			(* Постоянная часть передачи *)
			t_Msg.t_Id.u32_Id := 16#101;		(* Адрес пакета *)
			t_Msg.t_Id.u8_Xtd := 0;
			t_Msg.u8_Dlc      := 8;				(* Количество передаваемых байт *)
			t_Msg.au8_Data[0] := Can_buffer[CAN_TX_count+1];
			t_Msg.au8_Data[1] := Can_buffer[CAN_TX_count+2];
			t_Msg.au8_Data[2] := Can_buffer[CAN_TX_count+3];
			t_Msg.au8_Data[3] := Can_buffer[CAN_TX_count+4];
			t_Msg.au8_Data[4] := Can_buffer[CAN_TX_count+5];
			t_Msg.au8_Data[5] := Can_buffer[CAN_TX_count+6];
			t_Msg.au8_Data[6] := Can_buffer[CAN_TX_count+7];
			t_Msg.au8_Data[7] := Can_buffer[CAN_TX_count+8];
			fb_CanObjSendMsg(ou32_Handle:=TX, ot_Msg:=t_Msg, os16_Status=>s16_Return);
			CAN_TX_count:=CAN_TX_count+8;
		END_IF

END_IF
END_PROGRAM

(* POU CAN/Recieve, ST *)
PROGRAM Recieve
VAR
	s16_Return        	: INT;
	r_Msg			         : T_x_can_msg;
	fb_CanObjGetMsg   	: FB_x_can_obj_get_msg;
	fb_EepWrite  			: FB_x_eep_write;

	u16_Crc           	: UINT;
	fb_UtiCalcCrc16   	: FB_x_uti_calc_crc_16;
	i: WORD; (* Счетчик принятых по CAN пакетов в калибровке *)

	crc_given: UINT;
END_VAR
IF Flag_CAN THEN
			(* Что бы при ошибке чтения с CANa , при не изменении значений не произошо ложного срабатывания *)
			r_Msg.au8_Data[0]:=0;r_Msg.au8_Data[1]:=0;r_Msg.au8_Data[2]:=0;r_Msg.au8_Data[3]:=0;r_Msg.au8_Data[4]:=0;
			r_Msg.au8_Data[5]:=0;r_Msg.au8_Data[6]:=0;r_Msg.au8_Data[7]:=0;
			fb_CanObjGetMsg(ou32_Handle:=RX, ot_Msg=>r_Msg, os16_Status=>s16_Return);
			IF s16_Return = C_NO_ERR THEN

					(* Поступил запрос на передачу? *)
					IF	Flag_CAN_recieve=FALSE AND r_Msg.au8_Data[0] = 8 AND r_Msg.au8_Data[1] = 7 AND r_Msg.au8_Data[2] = 6 AND r_Msg.au8_Data[3] = 5 AND
						r_Msg.au8_Data[4] = 4 AND r_Msg.au8_Data[5] = 3 AND r_Msg.au8_Data[6] = 2 AND	r_Msg.au8_Data[7] = 1 THEN
						Flag_CAN_send:=TRUE;
					END_IF

					(* Поступил запрос на прием ? *)
					IF Flag_CAN_recieve = FALSE AND r_Msg.au8_Data[0] = 1 AND r_Msg.au8_Data[1] = 2 AND r_Msg.au8_Data[2] = 3 AND r_Msg.au8_Data[3] = 4 AND
						r_Msg.au8_Data[4] = 5 AND r_Msg.au8_Data[5] = 6 AND r_Msg.au8_Data[6] = 7 AND r_Msg.au8_Data[7] = 8 THEN

									Flag_CAN_recieve:=TRUE;
									i:=1;
					ELSIF i <= SIZEOF(Can_buffer)-7 THEN
											Can_buffer[i]:=r_Msg.au8_Data[0]; Can_buffer[i+1]:=r_Msg.au8_Data[1]; Can_buffer[i+2]:=r_Msg.au8_Data[2]; Can_buffer[i+3]:=r_Msg.au8_Data[3];
											Can_buffer[i+4]:=r_Msg.au8_Data[4]; Can_buffer[i+5]:=r_Msg.au8_Data[5]; Can_buffer[i+6]:=r_Msg.au8_Data[6]; Can_buffer[i+7]:=r_Msg.au8_Data[7];
											i:=i+8;
											IF i=SIZEOF(Can_buffer)+1 THEN
													Flag_CAN_recieve:= FALSE;
													(* Вычисляем CRC16 для массива передаваемых данных *)
													u16_Crc:=16#1D0F;
													fb_UtiCalcCrc16(ou32_Count:=SIZEOF(Can_buffer)-2, opu8_Data:=ADR(Can_buffer), ou16_Crc:=u16_Crc, os16_Status=>s16_Return);
													crc_given:= Can_buffer[SIZEOF(Can_buffer)]*256+Can_buffer[SIZEOF(Can_buffer)-1];
													IF crc_given =  u16_Crc THEN
															fb_EepWrite(ou32_Address:=0, ou32_Count:=SIZEOF(Can_buffer), opu8_Data:=ADR(Can_buffer), os16_Status=>s16_Return);
															Flag_CAN_Write:= TRUE;
													END_IF
											END_IF
					END_IF

			END_IF
END_IF
END_PROGRAM

(* Visualisation Calibrations/CALIBRATION_GAS_DIESEL
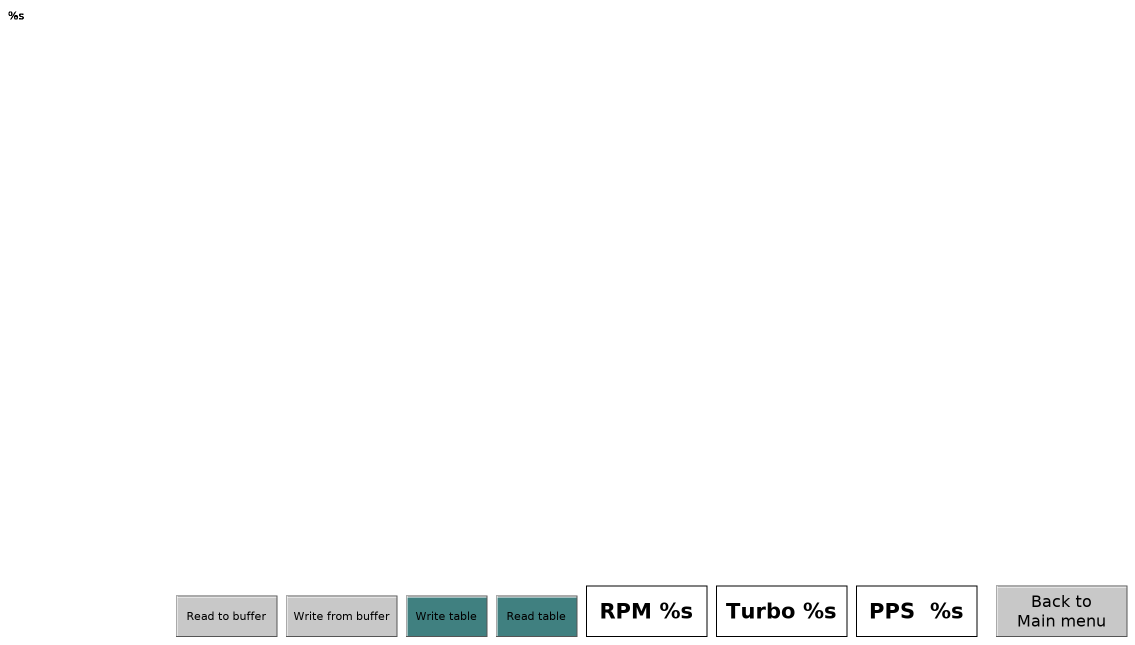
rectangle at (0,0)-(0,0): text "%s"; shows p.Turbo_table[1]; editable
rectangle at (0,0)-(0,0): text "%s"; shows p.Turbo_table[2]; editable
rectangle at (0,0)-(0,0): text "%s"; shows p.Turbo_table[3]; editable
rectangle at (0,0)-(0,0): text "%s"; shows p.Turbo_table[5]; editable
rectangle at (0,0)-(0,0): text "%s"; shows p.Turbo_table[4]; editable
rectangle at (0,0)-(0,0): text "%s"; shows p.Turbo_table[6]; editable
rectangle at (0,0)-(0,0): text "%s"; shows p.Turbo_table[8]; editable
rectangle at (0,0)-(0,0): text "%s"; shows p.Turbo_table[7]; editable
rectangle at (0,0)-(0,0): text "%s"; shows p.Turbo_table[9]; editable
rectangle at (0,0)-(0,0): text "%s"; shows p.Turbo_table[10]; editable
rectangle at (0,0)-(0,0): text "%s"; shows p.Turbo_table[13]; editable
rectangle at (0,0)-(0,0): text "%s"; shows p.Turbo_table[12]; editable
rectangle at (0,0)-(0,0): text "%s"; shows p.Turbo_table[11]; editable
button at (160,580)-(261,621): text "Read to buffer"; taps DFPRS_Change_Cal_Table.Red_cal_DF
button at (270,580)-(381,621): text "Write from buffer"; taps DFPRS_Change_Cal_Table.Write_cal_DF
button at (390,580)-(471,621): text "Write table"; taps DFPRS_Change_Cal_Table.Write_cal
button at (480,580)-(561,621): text "Read table"; taps DFPRS_Change_Cal_Table.Read_cal
rounded rectangle at (840,570)-(961,621): text "PPS  %s"; shows .PPS1
rounded rectangle at (570,570)-(691,621): text "RPM %s"; shows .RPM
rounded rectangle at (700,570)-(831,621): text "Turbo %s"; shows .Turbo_pressure
button at (980,570)-(1111,621): text "Back to / Main menu"; opens PLC_VISU
2 elements of other kinds (tables, trends, ...) not read
*)

(* Visualisation Check_parameters/CHECK_CURRENT
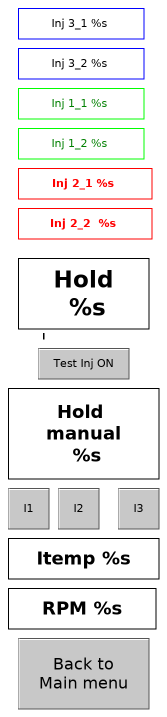
rounded rectangle at (1210,90)-(1336,121): text "Inj 1_1 %s"; shows .s32_Current_Inj1_1/1000
rounded rectangle at (1210,210)-(1344,241): text "Inj 2_2  %s"; shows .s32_Current_Inj2_2/1000
rounded rectangle at (1210,260)-(1341,331): text "Hold / %s"; shows .HOLD_time
rounded rectangle at (1210,10)-(1336,41): text "Inj 3_1 %s"; shows .s32_Current_Inj3_1/1000
rounded rectangle at (1210,130)-(1336,161): text "Inj 1_2 %s"; shows .s32_Current_Inj1_2/1000
rounded rectangle at (1210,170)-(1344,201): text "Inj 2_1 %s"; shows .s32_Current_Inj2_1/1000
rounded rectangle at (1210,50)-(1336,81): text "Inj 3_2 %s"; shows s32_Current_Inj3_2/1000
button at (1230,350)-(1321,381): text "Test Inj ON"; toggles .Flag_test_inj
rectangle at (1200,390)-(1351,481): text "Hold / manual / %s"; shows Act_control.Hold_manual; editable
button at (1200,490)-(1241,531): text "I1"; toggles .Flag_Inj1_ON
button at (1250,490)-(1291,531): text "I2"; toggles .Flag_Inj2_ON
button at (1310,490)-(1351,531): text "I3"; toggles .Flag_Inj3_ON
rounded rectangle at (1200,540)-(1351,581): text "Itemp %s"; shows .Injector_temp
rounded rectangle at (1200,590)-(1348,631): text "RPM %s"; shows .RPM
button at (1210,640)-(1341,711): text "Back to / Main menu"; opens PLC_VISU
1 more shapes without text or variables
1 elements of other kinds (tables, trends, ...) not read
*)

(* Visualisation Check_parameters/CHECK_EGT
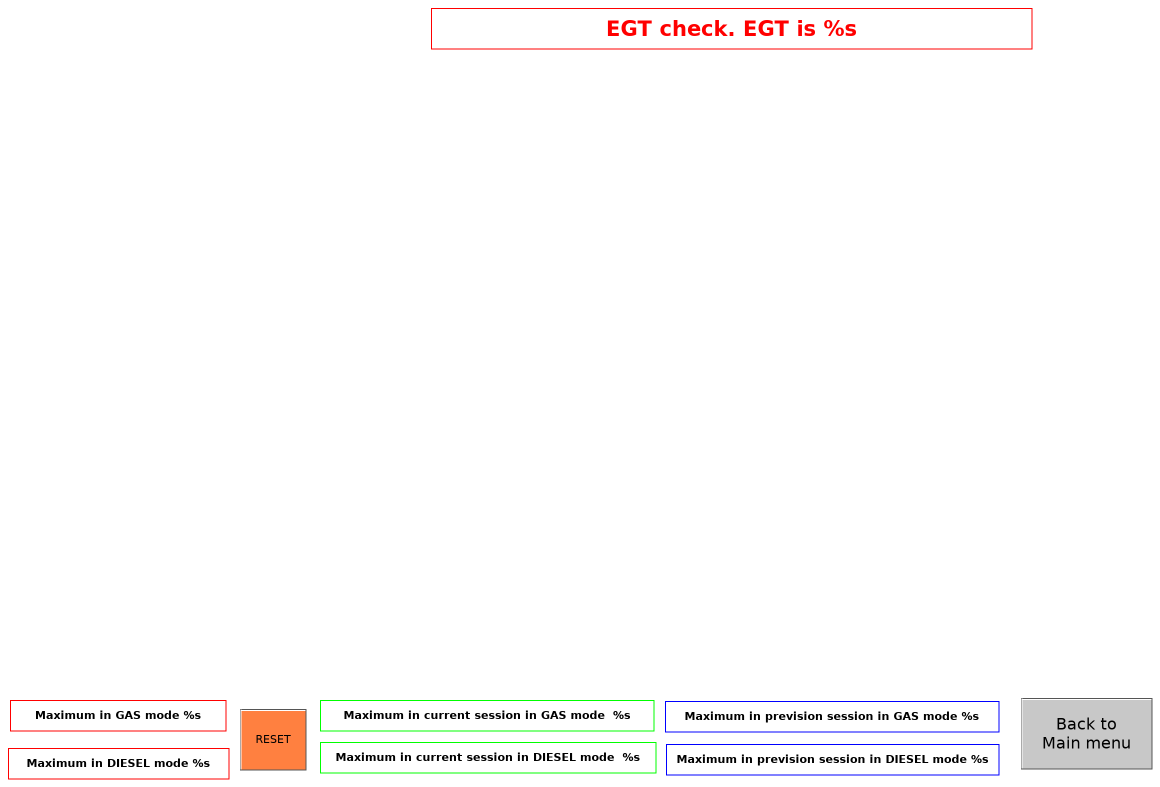
rounded rectangle at (9,702)-(225,733): text "Maximum in GAS mode %s"; shows .a.EGT_max_abs_GAS
rounded rectangle at (7,750)-(228,781): text "Maximum in DIESEL mode %s"; shows .a.EGT_max_abs_DIESEL
rounded rectangle at (665,746)-(998,777): text "Maximum in prevision session in DIESEL mode %s"; shows PLC_PRG.EGT_max_prev_sessions_DIESEL
rounded rectangle at (664,703)-(998,734): text "Maximum in prevision session in GAS mode %s"; shows PLC_PRG.EGT_max_prev_sessions_GAS
rounded rectangle at (319,702)-(653,733): text "Maximum in current session in GAS mode  %s"; shows .a.EGT_max_sessions_GAS
rounded rectangle at (319,744)-(655,775): text "Maximum in current session in DIESEL mode  %s"; shows .a.EGT_max_sessions_DIESEL
rounded rectangle at (430,10)-(1031,51): text "EGT check. EGT is %s"; shows .EGT
button at (239,711)-(305,772): text "RESET"; taps Get_EGT.Flag_EGT_reset
button at (1020,700)-(1151,771): text "Back to / Main menu"; opens PLC_VISU
1 elements of other kinds (tables, trends, ...) not read
*)

(* Visualisation Check_parameters/CHECK_INJ_TEMP
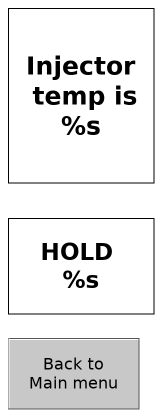
rounded rectangle at (1200,50)-(1346,225): text "Injector / temp is / %s"; shows .Injector_temp
rounded rectangle at (1200,260)-(1346,356): text "HOLD / %s"; shows .HOLD_time
button at (1200,380)-(1331,451): text "Back to / Main menu"; opens PLC_VISU
1 more shapes without text or variables
1 elements of other kinds (tables, trends, ...) not read
*)

(* Visualisation Check_parameters/CHECK_LOAD
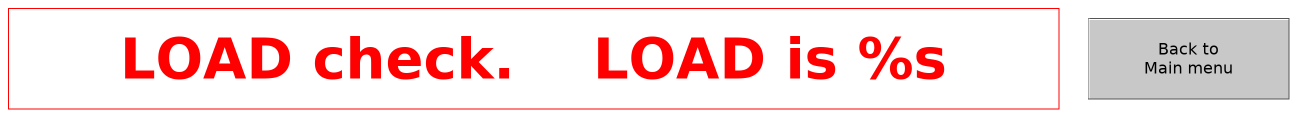
rounded rectangle at (30,10)-(1081,111): text "LOAD check.    LOAD is %s"; shows .Load
button at (1110,20)-(1311,101): text "Back to / Main menu"; opens PLC_VISU
1 elements of other kinds (tables, trends, ...) not read
*)

(* Visualisation FUEL
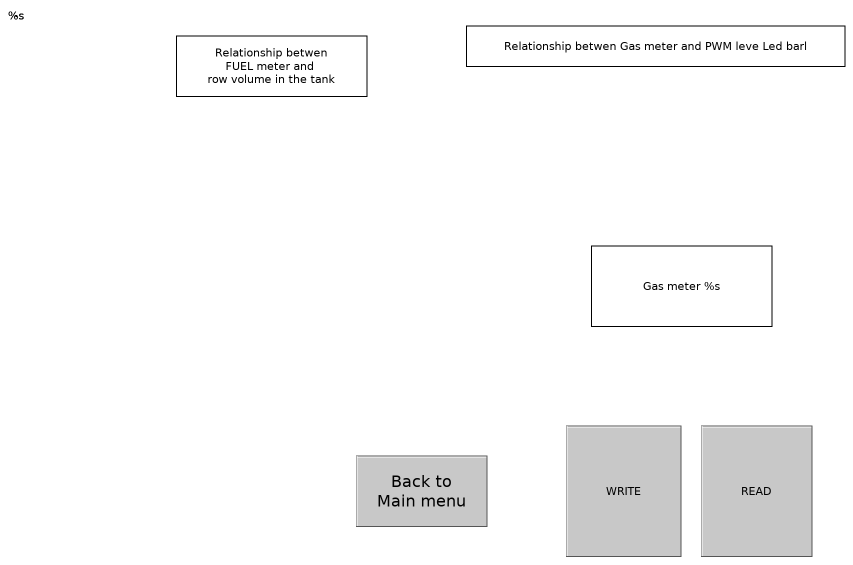
rounded rectangle at (450,10)-(829,51): text "Relationship betwen Gas meter and PWM leve Led barl"
rounded rectangle at (575,230)-(756,311): text "Gas meter %s"; shows .Gas_meter
rectangle at (0,0)-(0,0): text "%s"; shows p.LED_BAR_PWM[INDEX]; editable
rectangle at (0,0)-(0,0): text "%s"; shows p.Gas_meter_volume[INDEX]; editable
button at (550,410)-(665,541): text "WRITE"; taps DFPRS_Change_Cal_Table.Write_cal
button at (685,410)-(796,541): text "READ"; taps DFPRS_Change_Cal_Table.Read_cal
rounded rectangle at (160,20)-(351,81): text "Relationship betwen / FUEL meter and / row volume in the tank"
button at (340,440)-(471,511): text "Back to / Main menu"; opens PLC_VISU
2 elements of other kinds (tables, trends, ...) not read
*)

(* Visualisation MAIN_PRIBOR
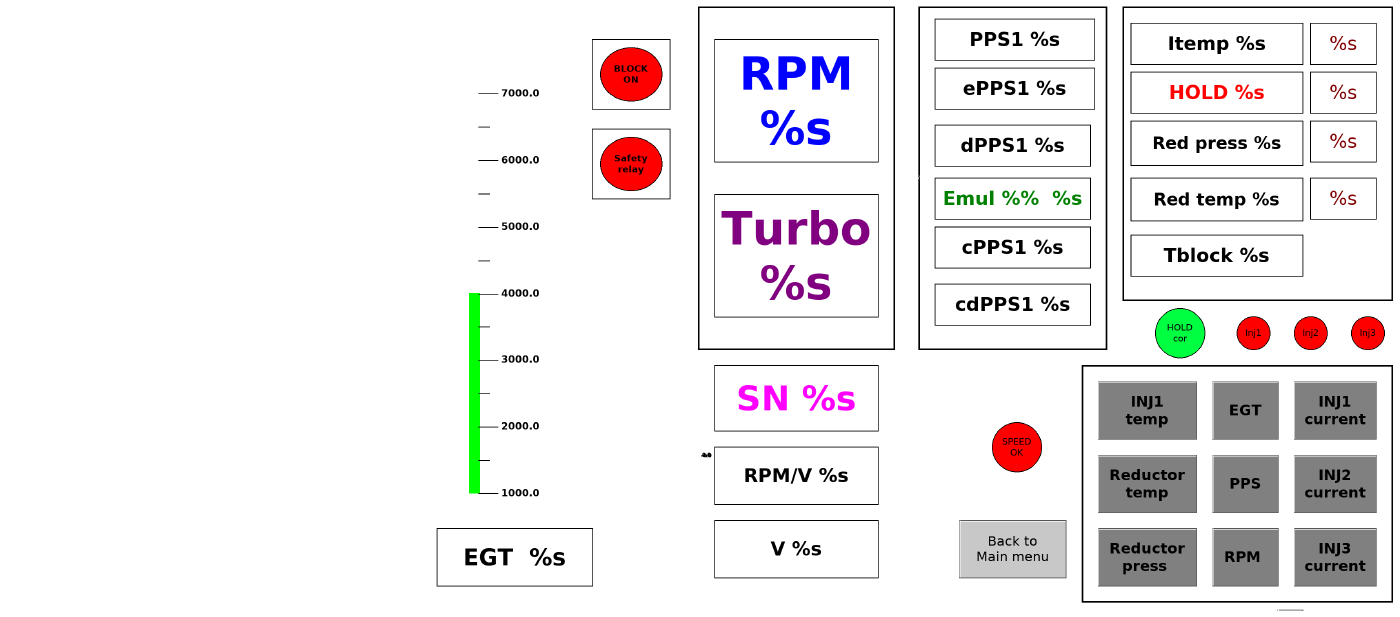
group at (370,220)-(371,221)
  rectangle at (0,0)-(1,1): text "{ExtendedElement},Visu\ElementDLL.ete,0,@Zeigerinstrument,200,180,0,0,255,255,255,0,,,%.1f,0,1,1,1,2,-4,4,0,0,0,0,0,0,0,-13,16,700,Arial,1,2,4000,5500,255,255,128,5500,6000,255,0,0,"
  rectangle at (1,92)-(23,108): text "-4.0"
  rectangle at (27,30)-(49,46): text "-2.0"
  rectangle at (91,4)-(109,20): text "0.0"
  rectangle at (153,30)-(171,46): text "2.0"
  rectangle at (179,92)-(197,108): text "4.0"
group at (370,560)-(371,561)
  rectangle at (0,0)-(1,1): text "{ExtendedElement},Visu\ElementDLL.ete,0,@Zeigerinstrument,200,180,0,0,255,255,255,0,,,%.1f,0,1,1,1,2,-4,4,0,0,0,0,0,0,0,-13,16,700,Arial,1,2,4000,5500,255,255,128,5500,6000,255,0,0,"
  rectangle at (1,92)-(23,108): text "-4.0"
  rectangle at (27,30)-(49,46): text "-2.0"
  rectangle at (91,4)-(109,20): text "0.0"
  rectangle at (153,30)-(171,46): text "2.0"
  rectangle at (179,92)-(197,108): text "4.0"
group at (60,80)-(171,618)
  rectangle at (0,0)-(1,1): text "{ExtendedElement},Visu\ElementDLL.ete,1,@Bargraph,111,538,0,1,0,EGT,,%.1f,500,1000,1000,7000,0,0,0,0,0,0,0,-13,16,700,Arial,0,255,0,255,0,0,1,6000,0,0,0,"
  rectangle at (18,268)-(30,502): alarm colour if (EGT) > 6000; top ((EGT * 1.0) - 4000)  * -0.078
  rectangle at (53,491)-(103,512): text "1000.0"
  rectangle at (53,413)-(103,434): text "2000.0"
  rectangle at (53,335)-(103,356): text "3000.0"
  rectangle at (53,258)-(103,279): text "4000.0"
  rectangle at (53,180)-(103,201): text "5000.0"
  rectangle at (53,102)-(103,123): text "6000.0"
  rectangle at (53,24)-(103,45): text "7000.0"
rounded rectangle at (890,220)-(1101,273): text "Red temp %s"; shows .Reductor_temp
rounded rectangle at (40,650)-(231,721): text "EGT  %s"; shows .EGT
rounded rectangle at (890,90)-(1101,141): text "HOLD %s"; shows .HOLD_time
rounded rectangle at (890,150)-(1101,205): text "Red press %s"; shows .Reductor_press
rounded rectangle at (890,30)-(1101,81): text "Itemp %s"; shows .Injector_temp
rounded rectangle at (650,25)-(846,76): text "PPS1 %s"; shows .PPS1
rounded rectangle at (650,85)-(846,136): text "ePPS1 %s"; shows .PPS1_emul
button at (990,650)-(1071,721): text "RPM"; toggles .Err_RPM
button at (990,470)-(1071,541): text "EGT"; toggles .Err_EGT
button at (850,560)-(971,631): text "Reductor / temp"; toggles .Err_Reductor_temp
button at (850,650)-(971,721): text "Reductor / press"; shows .Reductor_press; toggles .Err_Reductor_press
button at (1090,470)-(1191,541): text "INJ1 / current"; toggles .Err_Inj1
button at (1090,560)-(1191,631): text "INJ2 / current"; toggles .Err_Inj2
button at (850,470)-(971,541): text "INJ1 / temp"; toggles .Err_Inj_temp
button at (990,560)-(1071,631): text "PPS"; toggles .Err_PPS
button at (1090,650)-(1191,721): text "INJ3 / current"; toggles .Err_Inj3
rounded rectangle at (890,290)-(1101,341): text "Tblock %s"; shows .gs16_TempBoard
ellipse at (1020,390)-(1061,431): text "Inj1"; alarm colour if .Flag_Inj1_ON
ellipse at (1090,390)-(1131,431): text "Inj2"; alarm colour if .Flag_Inj2_ON
ellipse at (1160,390)-(1201,431): text "Inj3"; alarm colour if .Flag_Inj3_ON
rounded rectangle at (650,280)-(841,331): text "cPPS1 %s"; shows .cPPS1_emul
rounded rectangle at (650,350)-(841,401): text "cdPPS1 %s"; shows .PPS1-.cPPS1_emul
ellipse at (920,380)-(981,441): text "HOLD / cor"; alarm colour if .Flag_Inj_PWM_cor
button at (680,640)-(811,711): text "Back to / Main menu"; opens PLC_VISU
rounded rectangle at (650,155)-(841,206): text "dPPS1 %s"; shows .PPS1-.PPS1_emul
group at (230,160)-(326,246)
  ellipse at (10,10)-(86,76): text "Safety / relay"; alarm colour if .gq_Relay
group at (230,50)-(326,136)
  ellipse at (10,10)-(86,76): text "BLOCK / ON"; alarm colour if .Flag_ECU_ON
rounded rectangle at (380,240)-(581,391): text "Turbo / %s"; shows .Turbo_pressure
rounded rectangle at (380,50)-(581,201): text "RPM / %s"; shows .RPM
rounded rectangle at (380,550)-(581,621): text "RPM/V %s"; shows .Load
rectangle at (1110,30)-(1191,81): text "%s"; shows .p.Inj_temp_max
rectangle at (1110,90)-(1191,141): text "%s"; shows .p.Inj_MAX_hold_time/4
rectangle at (1110,150)-(1191,201): text "%s"; shows .p.Min_Reductor_press
rectangle at (1110,220)-(1191,271): text "%s"; shows .p.Reductor_temp_work
rounded rectangle at (650,220)-(841,271): text "Emul %%  %s"; shows 100-(.PPS1_emul*100)/.PPS1
rounded rectangle at (380,640)-(581,711): text "V %s"; shows .Speed
ellipse at (720,520)-(781,581): text "SPEED / OK"; alarm colour if Get_RPM_speed.Flag_speed_OK
rounded rectangle at (380,450)-(581,531): text "SN %s"; shows 1+(16-Act_control.z)
46 more shapes without text or variables
*)

(* Visualisation Calibrations/ONE_FUEL_CALIBRATION
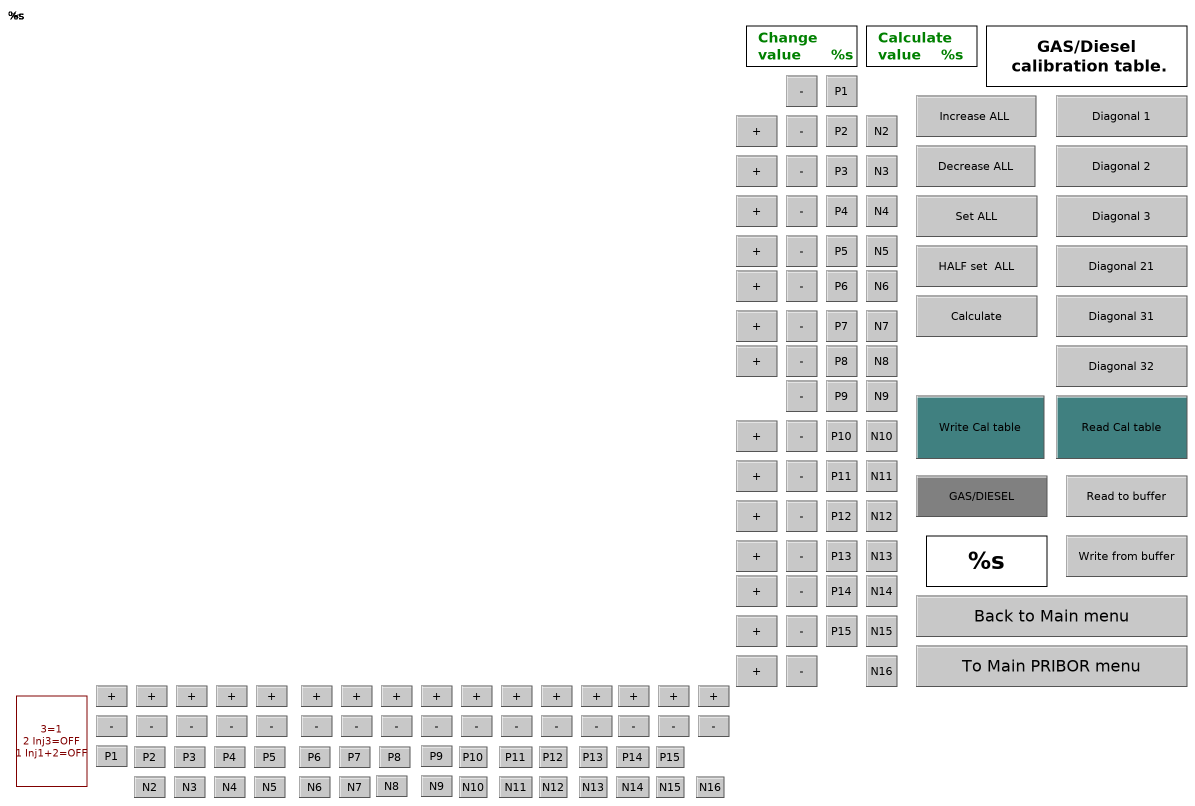
rectangle at (0,0)-(0,0): text "%s"; shows p.RPM_table[INDEX]; editable
rectangle at (0,0)-(0,0): text "%s"; shows p.Turbo_table[1]; editable
rectangle at (0,0)-(0,0): text "%s"; shows p.Turbo_table[2]; editable
rectangle at (0,0)-(0,0): text "%s"; shows p.Turbo_table[3]; editable
rectangle at (0,0)-(0,0): text "%s"; shows p.Turbo_table[4]; editable
rectangle at (0,0)-(0,0): text "%s"; shows p.Turbo_table[5]; editable
rectangle at (0,0)-(0,0): text "%s"; shows p.Turbo_table[6]; editable
rectangle at (0,0)-(0,0): text "%s"; shows p.Turbo_table[7]; editable
rectangle at (0,0)-(0,0): text "%s"; shows p.Turbo_table[8]; editable
rectangle at (0,0)-(0,0): text "%s"; shows p.Turbo_table[9]; editable
rectangle at (0,0)-(0,0): text "%s"; shows p.Turbo_table[10]; editable
rectangle at (0,0)-(0,0): text "%s"; shows p.Turbo_table[11]; editable
rectangle at (0,0)-(0,0): text "%s"; shows p.Turbo_table[12]; editable
rectangle at (0,0)-(0,0): text "%s"; shows p.Turbo_table[13]; editable
rectangle at (0,0)-(0,0): text "%s"; shows p.Turbo_table[14]; editable
rectangle at (0,0)-(0,0): text "%s"; shows p.Turbo_table[15]; editable
rectangle at (0,0)-(0,0): text "%s"; shows p.Turbo_table[16]; editable
button at (900,80)-(1020,121): text "Increase ALL"; taps DFPRS_Change_Cal_Table.ALL_plus
button at (900,130)-(1019,171): text "Decrease ALL"; taps DFPRS_Change_Cal_Table.ALL_minus
button at (1040,380)-(1171,443): text "Read Cal table"; taps DFPRS_Change_Cal_Table.Read_cal
button at (900,380)-(1028,443): text "Write Cal table"; taps DFPRS_Change_Cal_Table.Write_cal
button at (900,180)-(1021,221): text "Set ALL"; taps DFPRS_Change_Cal_Table.Set_ALL
button at (900,230)-(1021,271): text "HALF set  ALL"; taps DFPRS_Change_Cal_Table.HALF_set_ALL
button at (770,60)-(801,91): text "-"; taps DFPRS_Change_Cal_Table.RPM_Flag_minus_1
button at (720,100)-(761,131): text "+"; taps DFPRS_Change_Cal_Table.RPM_Flag_plus_2
button at (770,100)-(801,131): text "-"; taps DFPRS_Change_Cal_Table.RPM_Flag_minus_2
button at (810,100)-(841,131): text "P2"; taps DFPRS_Change_Cal_Table.RPM_Flag_CP_2
button at (720,140)-(761,171): text "+"; taps DFPRS_Change_Cal_Table.RPM_Flag_plus_3
button at (770,140)-(801,171): text "-"; taps DFPRS_Change_Cal_Table.RPM_Flag_minus_3
button at (810,140)-(841,171): text "P3"; taps DFPRS_Change_Cal_Table.RPM_Flag_CP_3
button at (720,180)-(761,211): text "+"; taps DFPRS_Change_Cal_Table.RPM_Flag_plus_4
button at (770,180)-(801,211): text "-"; taps DFPRS_Change_Cal_Table.RPM_Flag_minus_4
button at (810,180)-(841,211): text "P4"; taps DFPRS_Change_Cal_Table.RPM_Flag_CP_4
button at (720,220)-(761,251): text "+"; taps DFPRS_Change_Cal_Table.RPM_Flag_plus_5
button at (770,220)-(801,251): text "-"; taps DFPRS_Change_Cal_Table.RPM_Flag_minus_5
button at (810,220)-(841,251): text "P5"; taps DFPRS_Change_Cal_Table.RPM_Flag_CP_5
button at (720,255)-(761,286): text "+"; taps DFPRS_Change_Cal_Table.RPM_Flag_plus_6
button at (770,255)-(801,286): text "-"; taps DFPRS_Change_Cal_Table.RPM_Flag_minus_6
button at (810,255)-(841,286): text "P6"; taps DFPRS_Change_Cal_Table.RPM_Flag_CP_6
button at (720,295)-(761,326): text "+"; taps DFPRS_Change_Cal_Table.RPM_Flag_plus_7
button at (770,295)-(801,326): text "-"; taps DFPRS_Change_Cal_Table.RPM_Flag_minus_7
button at (810,295)-(841,326): text "P7"; taps DFPRS_Change_Cal_Table.RPM_Flag_CP_7
button at (720,330)-(761,361): text "+"; taps DFPRS_Change_Cal_Table.RPM_Flag_plus_8
button at (770,330)-(801,361): text "-"; taps DFPRS_Change_Cal_Table.RPM_Flag_minus_8
button at (810,330)-(841,361): text "P8"; taps DFPRS_Change_Cal_Table.RPM_Flag_CP_8
button at (80,670)-(111,691): text "+"; taps DFPRS_Change_Cal_Table.Turbo_Flag_plus_1
button at (80,700)-(111,721): text "-"; taps DFPRS_Change_Cal_Table.Turbo_Flag_minus_1
button at (120,670)-(151,691): text "+"; taps DFPRS_Change_Cal_Table.Turbo_Flag_plus_2
button at (120,700)-(151,721): text "-"; taps DFPRS_Change_Cal_Table.Turbo_Flag_minus_2
button at (118,731)-(149,752): text "P2"; taps DFPRS_Change_Cal_Table.Turbo_Flag_CP_2
button at (160,670)-(191,691): text "+"; taps DFPRS_Change_Cal_Table.Turbo_Flag_plus_3
button at (160,700)-(191,721): text "-"; taps DFPRS_Change_Cal_Table.Turbo_Flag_minus_3
button at (158,731)-(189,752): text "P3"; taps DFPRS_Change_Cal_Table.Turbo_Flag_CP_3
button at (200,670)-(231,691): text "+"; taps DFPRS_Change_Cal_Table.Turbo_Flag_plus_4
button at (200,700)-(231,721): text "-"; taps DFPRS_Change_Cal_Table.Turbo_Flag_minus_4
button at (198,731)-(229,752): text "P4"; taps DFPRS_Change_Cal_Table.Turbo_Flag_CP_4
button at (240,670)-(271,691): text "+"; taps DFPRS_Change_Cal_Table.Turbo_Flag_plus_5
button at (240,700)-(271,721): text "-"; taps DFPRS_Change_Cal_Table.Turbo_Flag_minus_5
button at (238,731)-(269,752): text "P5"; taps DFPRS_Change_Cal_Table.Turbo_Flag_CP_5
button at (285,670)-(316,691): text "+"; taps DFPRS_Change_Cal_Table.Turbo_Flag_plus_6
button at (285,700)-(316,721): text "-"; taps DFPRS_Change_Cal_Table.Turbo_Flag_minus_6
button at (283,731)-(314,752): text "P6"; taps DFPRS_Change_Cal_Table.Turbo_Flag_CP_6
button at (325,670)-(356,691): text "+"; taps DFPRS_Change_Cal_Table.Turbo_Flag_plus_7
button at (325,700)-(356,721): text "-"; taps DFPRS_Change_Cal_Table.Turbo_Flag_minus_7
button at (323,731)-(354,752): text "P7"; taps DFPRS_Change_Cal_Table.Turbo_Flag_CP_7
button at (365,670)-(396,691): text "+"; taps DFPRS_Change_Cal_Table.Turbo_Flag_plus_8
button at (365,700)-(396,721): text "-"; taps DFPRS_Change_Cal_Table.Turbo_Flag_minus_8
button at (363,731)-(394,752): text "P8"; taps DFPRS_Change_Cal_Table.Turbo_Flag_CP_8
rounded rectangle at (730,10)-(841,51): text "Change / value      %s"; shows DFPRS_Change_Cal_Table.Change_volume; editable 0..
rounded rectangle at (970,10)-(1171,71): text "GAS/Diesel / calibration table."
button at (1050,460)-(1171,501): text "Read to buffer"; taps DFPRS_Change_Cal_Table.red_cal2
button at (1050,520)-(1171,561): text "Write from buffer"; taps DFPRS_Change_Cal_Table.Write_cal2
button at (770,365)-(801,396): text "-"; taps DFPRS_Change_Cal_Table.RPM_Flag_minus_9
button at (720,405)-(761,436): text "+"; taps DFPRS_Change_Cal_Table.RPM_Flag_plus_10
button at (770,405)-(801,436): text "-"; taps DFPRS_Change_Cal_Table.RPM_Flag_minus_10
button at (810,405)-(841,436): text "P10"; taps DFPRS_Change_Cal_Table.RPM_Flag_CP_10
button at (720,445)-(761,476): text "+"; taps DFPRS_Change_Cal_Table.RPM_Flag_plus_11
button at (770,445)-(801,476): text "-"; taps DFPRS_Change_Cal_Table.RPM_Flag_minus_11
button at (810,445)-(841,476): text "P11"; taps DFPRS_Change_Cal_Table.RPM_Flag_CP_11
button at (720,485)-(761,516): text "+"; taps DFPRS_Change_Cal_Table.RPM_Flag_plus_12
button at (770,485)-(801,516): text "-"; taps DFPRS_Change_Cal_Table.RPM_Flag_minus_12
button at (810,485)-(841,516): text "P12"; taps DFPRS_Change_Cal_Table.RPM_Flag_CP_12
button at (720,525)-(761,556): text "+"; taps DFPRS_Change_Cal_Table.RPM_Flag_plus_13
button at (770,525)-(801,556): text "-"; taps DFPRS_Change_Cal_Table.RPM_Flag_minus_13
button at (810,525)-(841,556): text "P13"; taps DFPRS_Change_Cal_Table.RPM_Flag_CP_13
button at (810,365)-(841,396): text "P9"; taps DFPRS_Change_Cal_Table.RPM_Flag_CP_9
button at (405,670)-(436,691): text "+"; taps DFPRS_Change_Cal_Table.Turbo_Flag_plus_9
button at (405,700)-(436,721): text "-"; taps DFPRS_Change_Cal_Table.Turbo_Flag_minus_9
button at (445,670)-(476,691): text "+"; taps DFPRS_Change_Cal_Table.Turbo_Flag_plus_10
button at (445,700)-(476,721): text "-"; taps DFPRS_Change_Cal_Table.Turbo_Flag_minus_10
button at (443,731)-(471,752): text "P10"; taps DFPRS_Change_Cal_Table.Turbo_Flag_CP_10
button at (485,670)-(516,691): text "+"; taps DFPRS_Change_Cal_Table.Turbo_Flag_plus_11
button at (485,700)-(516,721): text "-"; taps DFPRS_Change_Cal_Table.Turbo_Flag_minus_11
button at (483,731)-(516,752): text "P11"; taps DFPRS_Change_Cal_Table.Turbo_Flag_CP_11
button at (525,670)-(556,691): text "+"; taps DFPRS_Change_Cal_Table.Turbo_Flag_plus_12
button at (525,700)-(556,721): text "-"; taps DFPRS_Change_Cal_Table.Turbo_Flag_minus_12
button at (523,731)-(551,752): text "P12"; taps DFPRS_Change_Cal_Table.Turbo_Flag_CP_12
button at (565,670)-(596,691): text "+"; taps DFPRS_Change_Cal_Table.Turbo_Flag_plus_13
button at (565,700)-(596,721): text "-"; taps DFPRS_Change_Cal_Table.Turbo_Flag_minus_13
button at (563,731)-(591,752): text "P13"; taps DFPRS_Change_Cal_Table.Turbo_Flag_CP_13
button at (405,730)-(436,751): text "P9"; taps DFPRS_Change_Cal_Table.Turbo_Flag_CP_9
rectangle at (0,680)-(71,771): text "3=1 / 2 Inj3=OFF / 1 Inj1+2=OFF"
button at (900,460)-(1031,501): text "GAS/DIESEL"; toggles DFPRS_Change_Cal_Table.Flag_cal_table_gas
rounded rectangle at (910,520)-(1031,571): text "%s"; shows DFPRS_Change_Cal_Table.Fuel_type
button at (900,280)-(1021,321): text "Calculate"; taps DFPRS_Change_Cal_Table.Calculate
rounded rectangle at (850,10)-(961,51): text "Calculate / value    %s"; shows DFPRS_Change_Cal_Table.Calculate_volume; editable 0..
button at (1040,80)-(1171,121): text "Diagonal 1"; taps DFPRS_Change_Cal_Table.Diagonal_1
button at (720,560)-(761,591): text "+"; taps DFPRS_Change_Cal_Table.RPM_Flag_plus_14
button at (770,560)-(801,591): text "-"; taps DFPRS_Change_Cal_Table.RPM_Flag_minus_14
button at (810,560)-(841,591): text "P14"; taps DFPRS_Change_Cal_Table.RPM_Flag_CP_14
button at (720,600)-(761,631): text "+"; taps DFPRS_Change_Cal_Table.RPM_Flag_plus_15
button at (770,600)-(801,631): text "-"; taps DFPRS_Change_Cal_Table.RPM_Flag_minus_15
button at (810,600)-(841,631): text "P15"; taps DFPRS_Change_Cal_Table.RPM_Flag_CP_15
button at (720,640)-(761,671): text "+"; taps DFPRS_Change_Cal_Table.RPM_Flag_plus_16
button at (770,640)-(801,671): text "-"; taps DFPRS_Change_Cal_Table.RPM_Flag_minus_16
button at (810,60)-(841,91): text "P1"; taps DFPRS_Change_Cal_Table.RPM_Flag_CP_1
button at (850,100)-(881,131): text "N2"; taps DFPRS_Change_Cal_Table.RPM_Flag_CN_2
button at (850,140)-(881,171): text "N3"; taps DFPRS_Change_Cal_Table.RPM_Flag_CN_3
button at (850,180)-(881,211): text "N4"; taps DFPRS_Change_Cal_Table.RPM_Flag_CN_4
button at (850,220)-(881,251): text "N5"; taps DFPRS_Change_Cal_Table.RPM_Flag_CN_5
button at (850,255)-(881,286): text "N6"; taps DFPRS_Change_Cal_Table.RPM_Flag_CN_6
button at (850,295)-(881,326): text "N7"; taps DFPRS_Change_Cal_Table.RPM_Flag_CN_7
button at (850,330)-(881,361): text "N8"; taps DFPRS_Change_Cal_Table.RPM_Flag_CN_8
button at (850,405)-(881,436): text "N10"; taps DFPRS_Change_Cal_Table.RPM_Flag_CN_10
button at (850,445)-(881,476): text "N11"; taps DFPRS_Change_Cal_Table.RPM_Flag_CN_11
button at (850,485)-(881,516): text "N12"; taps DFPRS_Change_Cal_Table.RPM_Flag_CN_12
button at (850,525)-(881,556): text "N13"; taps DFPRS_Change_Cal_Table.RPM_Flag_CN_13
button at (850,365)-(881,396): text "N9"; taps DFPRS_Change_Cal_Table.RPM_Flag_CN_9
button at (850,560)-(881,591): text "N14"; taps DFPRS_Change_Cal_Table.RPM_Flag_CN_14
button at (850,600)-(881,631): text "N15"; taps DFPRS_Change_Cal_Table.RPM_Flag_CN_15
button at (850,640)-(881,671): text "N16"; taps DFPRS_Change_Cal_Table.RPM_Flag_CN_16
button at (1040,130)-(1171,171): text "Diagonal 2"; taps DFPRS_Change_Cal_Table.Diagonal_2
button at (1040,180)-(1171,221): text "Diagonal 3"; taps DFPRS_Change_Cal_Table.Diagonal_3
button at (1040,230)-(1171,271): text "Diagonal 21"; taps DFPRS_Change_Cal_Table.Diagonal_21
button at (1040,280)-(1171,321): text "Diagonal 31"; taps DFPRS_Change_Cal_Table.Diagonal_31
button at (900,580)-(1171,621): text "Back to Main menu"; opens PLC_VISU
button at (900,630)-(1171,671): text "To Main PRIBOR menu"; opens MAIN_PRIBOR
button at (602,670)-(633,691): text "+"; taps DFPRS_Change_Cal_Table.Turbo_Flag_plus_14
button at (602,700)-(633,721): text "-"; taps DFPRS_Change_Cal_Table.Turbo_Flag_minus_14
button at (600,731)-(633,752): text "P14"; taps DFPRS_Change_Cal_Table.Turbo_Flag_CP_14
button at (642,670)-(673,691): text "+"; taps DFPRS_Change_Cal_Table.Turbo_Flag_plus_15
button at (642,700)-(673,721): text "-"; taps DFPRS_Change_Cal_Table.Turbo_Flag_minus_15
button at (640,731)-(668,752): text "P15"; taps DFPRS_Change_Cal_Table.Turbo_Flag_CP_15
button at (682,670)-(713,691): text "+"; taps DFPRS_Change_Cal_Table.Turbo_Flag_plus_16
button at (682,700)-(713,721): text "-"; taps DFPRS_Change_Cal_Table.Turbo_Flag_minus_16
button at (80,730)-(111,751): text "P1"; taps DFPRS_Change_Cal_Table.Turbo_Flag_CP_1
button at (118,761)-(149,782): text "N2"; taps DFPRS_Change_Cal_Table.Turbo_Flag_CN_2
button at (158,761)-(189,782): text "N3"; taps DFPRS_Change_Cal_Table.Turbo_Flag_CN_3
button at (198,761)-(229,782): text "N4"; taps DFPRS_Change_Cal_Table.Turbo_Flag_CN_4
button at (238,761)-(269,782): text "N5"; taps DFPRS_Change_Cal_Table.Turbo_Flag_CN_5
button at (283,761)-(314,782): text "N6"; taps DFPRS_Change_Cal_Table.Turbo_Flag_CN_6
button at (323,761)-(354,782): text "N7"; taps DFPRS_Change_Cal_Table.Turbo_Flag_CN_7
button at (360,760)-(391,781): text "N8"; taps DFPRS_Change_Cal_Table.Turbo_Flag_CN_8
button at (443,761)-(471,782): text "N10"; taps DFPRS_Change_Cal_Table.Turbo_Flag_CN_10
button at (483,761)-(516,782): text "N11"; taps DFPRS_Change_Cal_Table.Turbo_Flag_CN_11
button at (523,761)-(551,782): text "N12"; taps DFPRS_Change_Cal_Table.Turbo_Flag_CN_12
button at (563,761)-(591,782): text "N13"; taps DFPRS_Change_Cal_Table.Turbo_Flag_CN_13
button at (405,760)-(436,781): text "N9"; taps DFPRS_Change_Cal_Table.Turbo_Flag_CN_9
button at (600,761)-(633,782): text "N14"; taps DFPRS_Change_Cal_Table.Turbo_Flag_CN_14
button at (640,761)-(668,782): text "N15"; taps DFPRS_Change_Cal_Table.Turbo_Flag_CN_15
button at (680,761)-(708,782): text "N16"; taps DFPRS_Change_Cal_Table.Turbo_Flag_CN_16
button at (1040,330)-(1171,371): text "Diagonal 32"; taps DFPRS_Change_Cal_Table.Diagonal_32
*)

(* Visualisation PLC_VISU
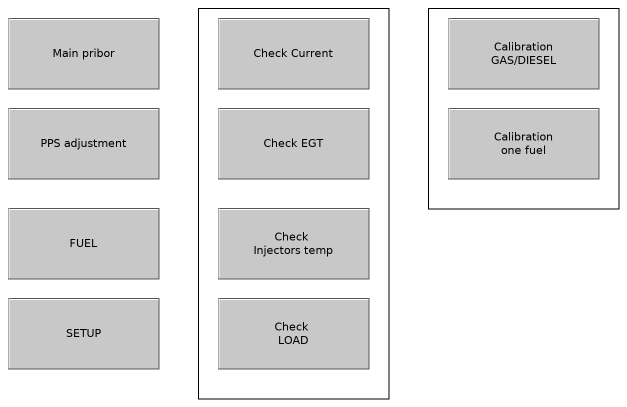
button at (40,30)-(191,101): text "Main pribor"; opens MAIN_PRIBOR
button at (250,30)-(401,101): text "Check Current"; opens CHECK_CURRENT
button at (250,120)-(401,191): text "Check EGT"; opens CHECK_EGT
button at (250,220)-(401,291): text "Check / Injectors temp"; opens CHECK_INJ_TEMP
button at (480,30)-(631,101): text "Calibration / GAS/DIESEL"; opens CALIBRATION_GAS_DIESEL
button at (480,120)-(631,191): text "Calibration / one fuel"; opens ONE_FUEL_CALIBRATION
button at (40,120)-(191,191): text "PPS adjustment"; opens PPS_PWM_adjustment
button at (40,220)-(191,291): text "FUEL"; opens FUEL
button at (250,310)-(401,381): text "Check / LOAD"; opens CHECK_Load
button at (40,310)-(191,381): text "SETUP"; opens SETUP
2 more shapes without text or variables
*)

(* Visualisation PPS_PWM_ADJUSTMENT
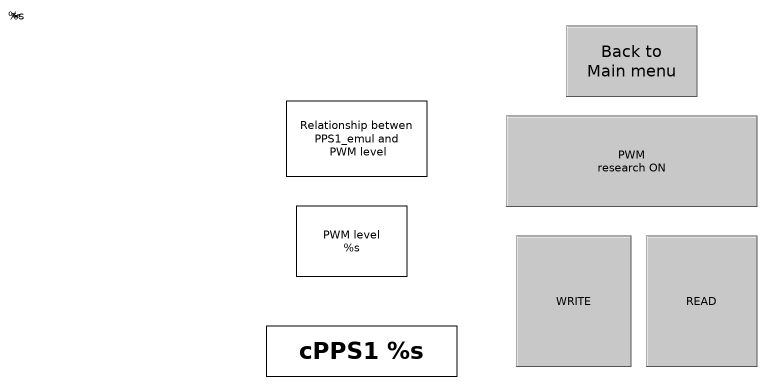
button at (490,100)-(741,191): text "PWM / research ON"; toggles .Flag_PWM_researh
button at (500,220)-(615,351): text "WRITE"; taps DFPRS_Change_Cal_Table.Write_cal
button at (630,220)-(741,351): text "READ"; taps DFPRS_Change_Cal_Table.Read_cal
rounded rectangle at (270,85)-(411,161): text "Relationship betwen / PPS1_emul and / PWM level"
rounded rectangle at (280,190)-(391,261): text "PWM level / %s"; shows Act_control.PPS_PWM; editable
rectangle at (0,0)-(0,0): text "%s"; shows p.PPS1_emul_PWM[INDEX]; editable
rectangle at (0,0)-(0,0): text "%s"; shows p.PPS_table[INDEX]; editable
rounded rectangle at (250,310)-(441,361): text "cPPS1 %s"; shows .cPPS1_emul
button at (550,10)-(681,81): text "Back to / Main menu"; opens PLC_VISU
rectangle at (0,0)-(0,0): text "%s"; shows p.Load_table[INDEX]; editable
rectangle at (0,0)-(0,0): text "%s"; shows p.GAS_Load_table[INDEX]; editable
rectangle at (0,0)-(0,0): text "%s"; shows p.DIESEL_Load_table[INDEX]; editable
*)

(* Visualisation SETUP
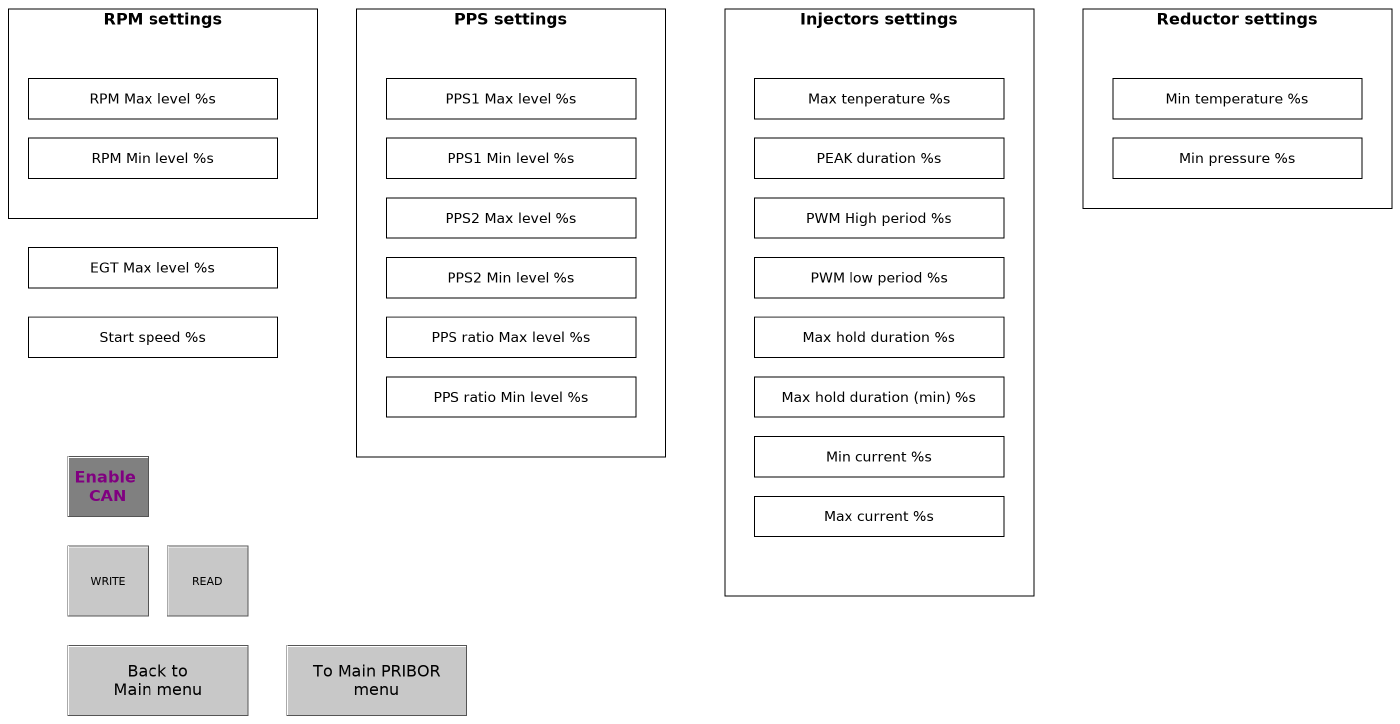
rounded rectangle at (1100,90)-(1411,291): text "Reductor settings"
rounded rectangle at (20,90)-(331,301): text "RPM settings"
button at (80,540)-(161,601): text "Enable / CAN"; toggles .Flag_CAN
rounded rectangle at (40,330)-(291,371): text "EGT Max level %s"; shows .p.EGT_max; editable
button at (180,630)-(261,701): text "READ"; taps DFPRS_Change_Cal_Table.Read_cal
button at (80,630)-(161,701): text "WRITE"; taps DFPRS_Change_Cal_Table.Write_cal
button at (80,730)-(261,801): text "Back to / Main menu"; opens PLC_VISU
rounded rectangle at (40,160)-(291,201): text "RPM Max level %s"; shows .p.RPM_max; editable
rounded rectangle at (40,220)-(291,261): text "RPM Min level %s"; shows .p.RPM_min; editable
rounded rectangle at (1130,160)-(1381,201): text "Min temperature %s"; shows .p.Reductor_temp_work; editable
rounded rectangle at (1130,220)-(1381,261): text "Min pressure %s"; shows .p.Min_Reductor_press; editable
rounded rectangle at (370,90)-(681,541): text "PPS settings"
rounded rectangle at (400,160)-(651,201): text "PPS1 Max level %s"; shows .p.PPS1_max; editable
rounded rectangle at (400,220)-(651,261): text "PPS1 Min level %s"; shows .p.PPS1_min; editable
rounded rectangle at (400,280)-(651,321): text "PPS2 Max level %s"; shows .p.PPS2_max; editable
rounded rectangle at (400,340)-(651,381): text "PPS2 Min level %s"; shows .p.PPS2_min; editable
rounded rectangle at (400,400)-(651,441): text "PPS ratio Max level %s"; shows .p.PPS_ratio_max; editable
rounded rectangle at (400,460)-(651,501): text "PPS ratio Min level %s"; shows .p.PPS_ratio_min; editable
rounded rectangle at (740,90)-(1051,681): text "Injectors settings"; tooltip Значения настроек для инжекторов надо менять очень осторожно. И хорошо представлять себя последствия.
rounded rectangle at (770,400)-(1021,441): text "Max hold duration %s"; shows .p.Inj_MAX_hold_time; tooltip Абсолютное ограничение максимальной длительности тока удержания. Задается в циклах по 250 мкс. HOLD 1 мс =4*250 мкс; editable
rounded rectangle at (770,460)-(1021,501): text "Max hold duration (min) %s"; shows .p.Inj_MAX_hold_time_min; tooltip Ограничение максимальной длительности тока удержания для первых трех значений RPM и Turbo Задается в циклах по 250 мкс. HOLD 1 мс =4*250 мкс; editable
button at (300,730)-(481,801): text "To Main PRIBOR / menu"; opens MAIN_PRIBOR
rounded rectangle at (770,340)-(1021,381): text "PWM low period %s"; shows .p.Inj_Low_period; tooltip Задание скважности PWM форсунок ( соотношение кол-ва ЦИКЛОВ низкого сигнала к одному ВЫСОКОМУ циклу ), подбирается имперически по условию соблюдения уровня холдового тока на форсунке; editable
rounded rectangle at (770,280)-(1021,321): text "PWM High period %s"; shows .p.Inj_High_period; tooltip Задание скважности PWM форсунок ( соотношение кол-ва ЦИКЛОВ низкого сигнала к одному ВЫСОКОМУ циклу ), подбирается имперически по условию соблюдения уровня холдового тока на форсунке; editable
rounded rectangle at (770,220)-(1021,261): text "PEAK duration %s"; shows .p.Inj_peak_curent_cycle; tooltip Количество циклов по 250 мкс для генерирования пикового импульса открытия форсунки; editable
rounded rectangle at (770,160)-(1021,201): text "Max tenperature %s"; shows .p.Inj_temp_max; tooltip Максимальный ток в микроамперах, протекающий через терморезистор на рейке; editable
rounded rectangle at (770,520)-(1021,561): text "Min current %s"; shows .p.Min_inj_current; tooltip Минимальный длительный ток через форсунки; editable
rounded rectangle at (770,580)-(1021,621): text "Max current %s"; shows .p.Max_inj_current; tooltip Максимальный длительный ток через форсунки; editable
rounded rectangle at (40,400)-(291,441): text "Start speed %s"; shows .p.Speed_limit; editable
*)
